// Mitsubishi GX Works2 project: LINEB-070924   PLC: Q26UDV

// task Task_01 (event TRUE, interval 0, priority 31): POU_01
// task temp_system (event TRUE, interval 0, priority 31): temp_system
// task comparater (event TRUE, interval 0, priority 31): comparater
// task Display (event TRUE, interval 0, priority 31): Display
// task cover_system (event TRUE, interval 0, priority 31): cover_system
// task input (event TRUE, interval 0, priority 31): input
// task output (event TRUE, interval 0, priority 31): output
// task payanak (event TRUE, interval 0, priority 31): 
// task pump_by_p_tongg (event TRUE, interval 0, priority 31): pump_by_p_tongg
// task rotation (event TRUE, interval 0, priority 31): rotation
// task lift (event TRUE, interval 0, priority 31): lift
// task blower (event TRUE, interval 0, priority 31): blower
// task carrier_move (event TRUE, interval 0, priority 31): carrier_move
// task door (event TRUE, interval 0, priority 31): door
// task lift_door_step (event TRUE, interval 0, priority 31): lift_door_step
// task Bit_Moniter_B (event TRUE, interval 0, priority 31): Bit_Moniter_B
// task input_conveyer (event TRUE, interval 0, priority 31): conveyer_input
// task coveyor_system (event TRUE, interval 0, priority 31): coveyor_system
// task convetor_output (event TRUE, interval 0, priority 31): conveyor_output
// task Scrubber (event TRUE, interval 0, priority 31): Scrubber
// task busket (event TRUE, interval 0, priority 31): busket
// task enter_line (event TRUE, interval 0, priority 31): enter_line
// task oven (event TRUE, interval 0, priority 31): oven
// task request_data (event TRUE, interval 0, priority 31): request_data
// task shower (event TRUE, interval 0, priority 31): shower
// task data_exchage (event TRUE, interval 0, priority 31): data_exchage
// task Alarm (event TRUE, interval 0, priority 31): Alarm
// task tower_lamp (event TRUE, interval 0, priority 31): tower_lamp
// task busker_step (event TRUE, interval 0, priority 31): busker_step
// task bit_monitor (event TRUE, interval 0, priority 31): bit_monitor
// task unload (event TRUE, interval 0, priority 31): unload
// task water_supply (event TRUE, interval 0, priority 31): water_supply
// task carrier_reset (event TRUE, interval 0, priority 31): carrier_reset
// task safty (event TRUE, interval 0, priority 31): safty
// task send_to_c (event TRUE, interval 0, priority 31): send_to_c
// task next_cap_step (event TRUE, interval 0, priority 31): next_cap_step
// task sent_to_c_key (event TRUE, interval 0, priority 31): sent_to_c_key
// task tank_time_B (event TRUE, interval 0, priority 31): tank_time_B
// task receive_c (event TRUE, interval 0, priority 31): receive_c
// task carrier_01 (event TRUE, interval 0, priority 31): carrier_01
// task carrier_02 (event TRUE, interval 0, priority 31): carrier_02
// task carrier_03 (event TRUE, interval 0, priority 31): carrier_03

PROGRAM Alarm
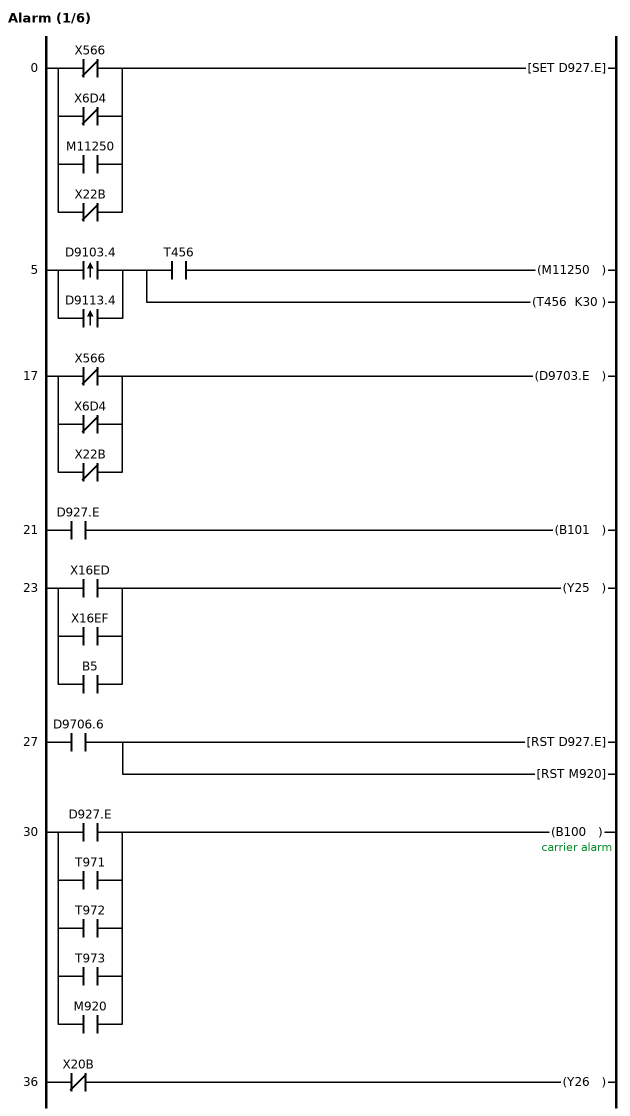
0     LDI     X566
      ORI     X6D4
      OR      M11250
      ORI     X22B
      SET     D927.E
5     LDP     D9103.4
      ORP     D9113.4
      MPS
      AND     T456
      OUT     M11250
      MPP
      OUT     T456 K30
17    LDI     X566
      ORI     X6D4
      ORI     X22B
      OUT     D9703.E
21    LD      D927.E
      OUT     B101
23    LD      X16ED
      OR      X16EF
      OR      B5
      OUT     Y25
27    LD      D9706.6
      RST     D927.E
      RST     M920
30    LD      D927.E
      OR      T971
      OR      T972
      OR      T973
      OR      M920
      OUT     B100  ; carrier alarm
36    LDI     X20B
      OUT     Y26
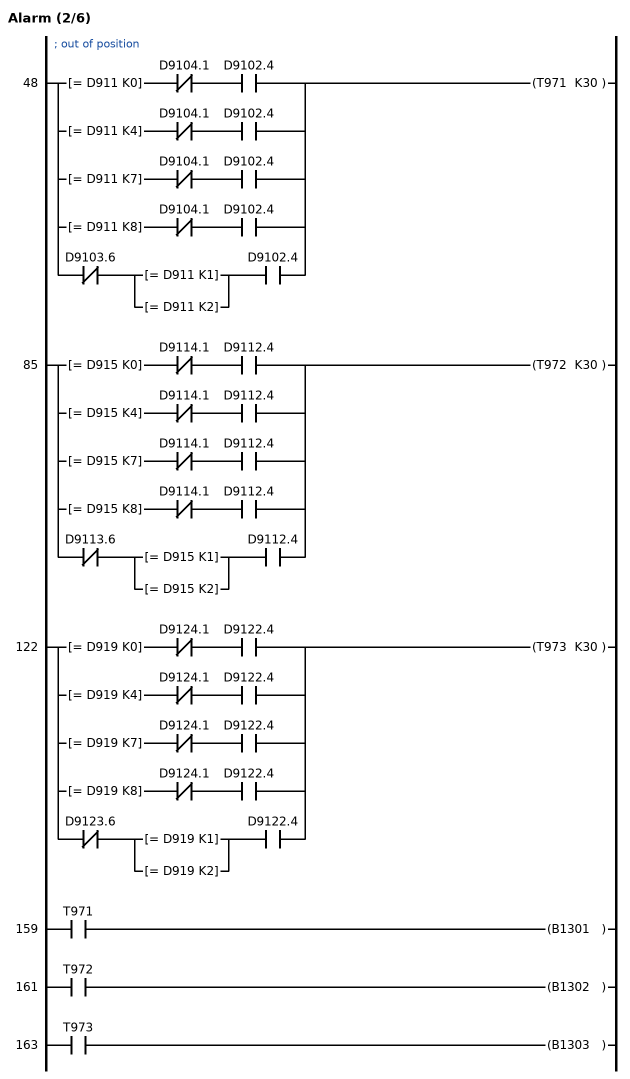
; out of position
48    LD=     D911 K0
      ANI     D9104.1
      AND     D9102.4
      LD=     D911 K4
      ANI     D9104.1
      AND     D9102.4
      ORB
      LD=     D911 K7
      ANI     D9104.1
      AND     D9102.4
      ORB
      LD=     D911 K8
      ANI     D9104.1
      AND     D9102.4
      ORB
      LDI     D9103.6
      LD=     D911 K1
      OR=     D911 K2
      ANB
      AND     D9102.4
      ORB
      OUT     T971 K30
85    LD=     D915 K0
      ANI     D9114.1
      AND     D9112.4
      LD=     D915 K4
      ANI     D9114.1
      AND     D9112.4
      ORB
      LD=     D915 K7
      ANI     D9114.1
      AND     D9112.4
      ORB
      LD=     D915 K8
      ANI     D9114.1
      AND     D9112.4
      ORB
      LDI     D9113.6
      LD=     D915 K1
      OR=     D915 K2
      ANB
      AND     D9112.4
      ORB
      OUT     T972 K30
122   LD=     D919 K0
      ANI     D9124.1
      AND     D9122.4
      LD=     D919 K4
      ANI     D9124.1
      AND     D9122.4
      ORB
      LD=     D919 K7
      ANI     D9124.1
      AND     D9122.4
      ORB
      LD=     D919 K8
      ANI     D9124.1
      AND     D9122.4
      ORB
      LDI     D9123.6
      LD=     D919 K1
      OR=     D919 K2
      ANB
      AND     D9122.4
      ORB
      OUT     T973 K30
159   LD      T971
      OUT     B1301
161   LD      T972
      OUT     B1302
163   LD      T973
      OUT     B1303
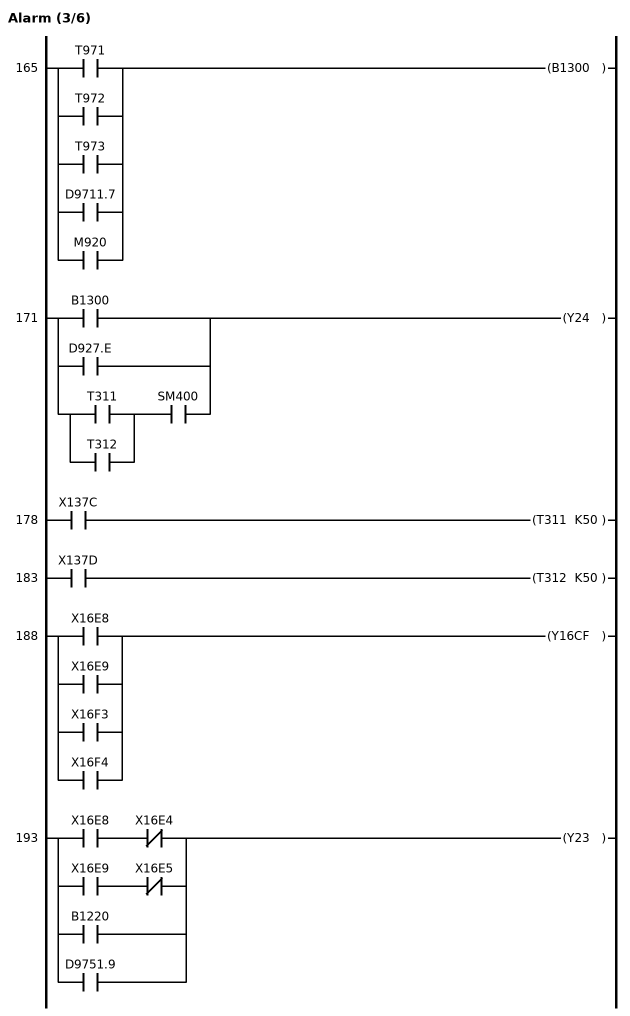
165   LD      T971
      OR      T972
      OR      T973
      OR      D9711.7
      OR      M920
      OUT     B1300
171   LD      B1300
      OR      D927.E
      LD      T311
      OR      T312
      AND     SM400
      ORB
      OUT     Y24
178   LD      X137C
      OUT     T311 K50
183   LD      X137D
      OUT     T312 K50
188   LD      X16E8
      OR      X16E9
      OR      X16F3
      OR      X16F4
      OUT     Y16CF
193   LD      X16E8
      ANI     X16E4
      LD      X16E9
      ANI     X16E5
      ORB
      OR      B1220
      OR      D9751.9
      OUT     Y23
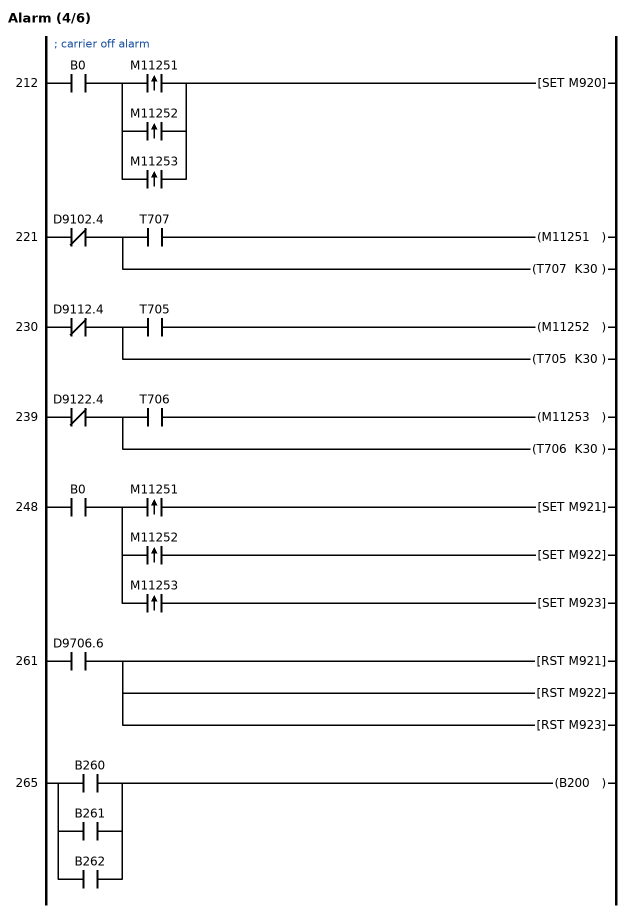
; carrier off alarm
212   LD      B0
      LDP     M11251
      ORP     M11252
      ORP     M11253
      ANB
      SET     M920
221   LDI     D9102.4
      MPS
      AND     T707
      OUT     M11251
      MPP
      OUT     T707 K30
230   LDI     D9112.4
      MPS
      AND     T705
      OUT     M11252
      MPP
      OUT     T705 K30
239   LDI     D9122.4
      MPS
      AND     T706
      OUT     M11253
      MPP
      OUT     T706 K30
248   LD      B0
      MPS
      ANDP    M11251
      SET     M921
      MRD
      ANDP    M11252
      SET     M922
      MPP
      ANDP    M11253
      SET     M923
261   LD      D9706.6
      RST     M921
      RST     M922
      RST     M923
265   LD      B260
      OR      B261
      OR      B262
      OUT     B200
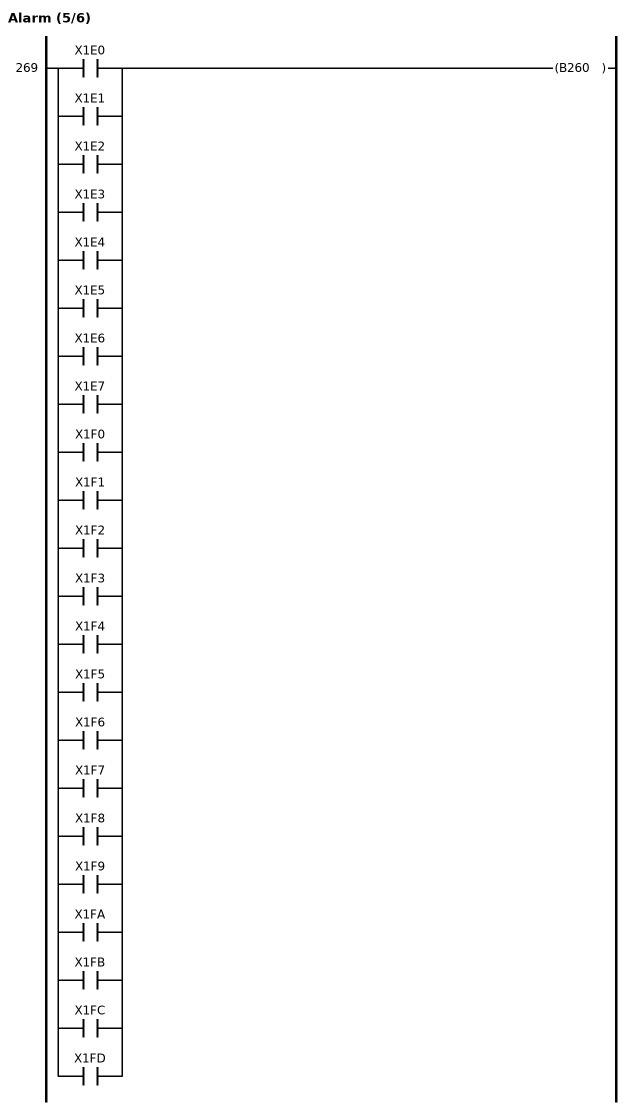
269   LD      X1E0
      OR      X1E1
      OR      X1E2
      OR      X1E3
      OR      X1E4
      OR      X1E5
      OR      X1E6
      OR      X1E7
      OR      X1F0
      OR      X1F1
      OR      X1F2
      OR      X1F3
      OR      X1F4
      OR      X1F5
      OR      X1F6
      OR      X1F7
      OR      X1F8
      OR      X1F9
      OR      X1FA
      OR      X1FB
      OR      X1FC
      OR      X1FD
      OUT     B260
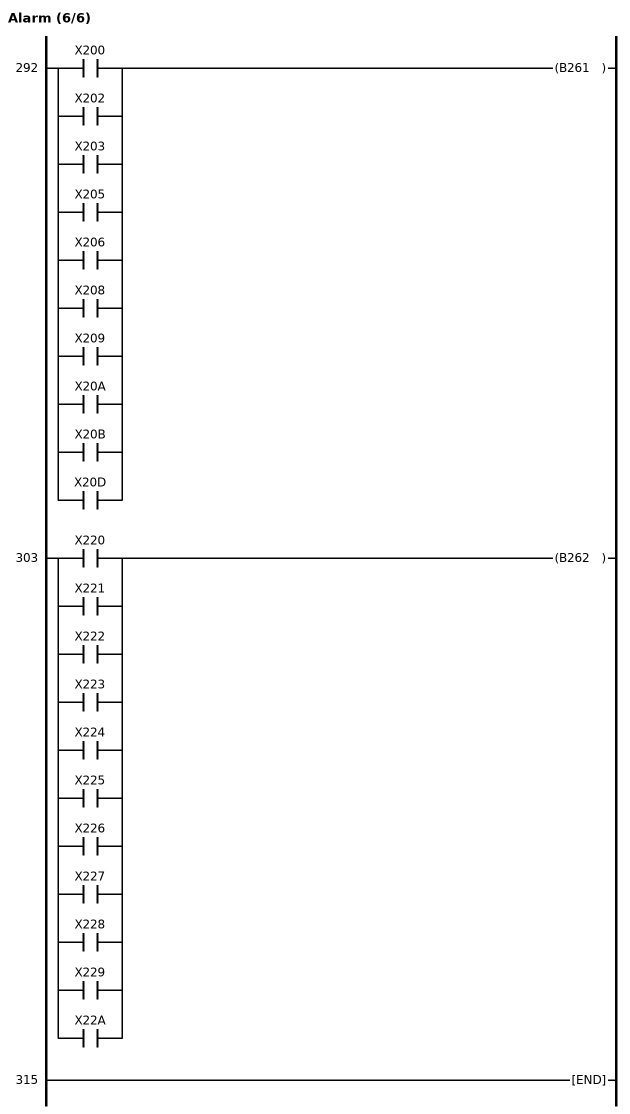
292   LD      X200
      OR      X202
      OR      X203
      OR      X205
      OR      X206
      OR      X208
      OR      X209
      OR      X20A
      OR      X20B
      OR      X20D
      OUT     B261
303   LD      X220
      OR      X221
      OR      X222
      OR      X223
      OR      X224
      OR      X225
      OR      X226
      OR      X227
      OR      X228
      OR      X229
      OR      X22A
      OUT     B262
315   END
END_PROGRAM

PROGRAM Bit_Moniter_B
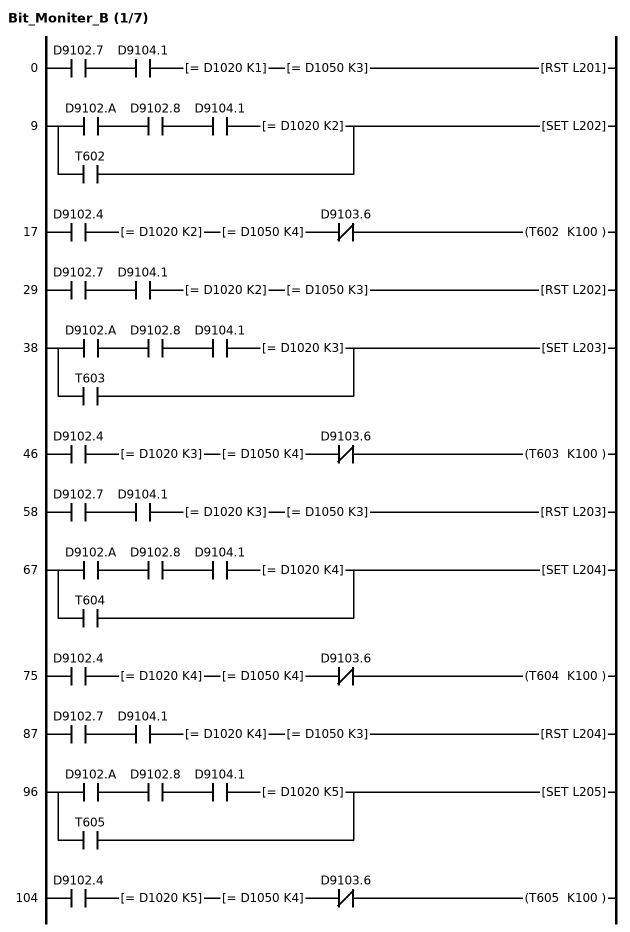
0     LD      D9102.7
      AND     D9104.1
      AND=    D1020 K1
      AND=    D1050 K3
      RST     L201
9     LD      D9102.A
      AND     D9102.8
      AND     D9104.1
      AND=    D1020 K2
      OR      T602
      SET     L202
17    LD      D9102.4
      AND=    D1020 K2
      AND=    D1050 K4
      ANI     D9103.6
      OUT     T602 K100
29    LD      D9102.7
      AND     D9104.1
      AND=    D1020 K2
      AND=    D1050 K3
      RST     L202
38    LD      D9102.A
      AND     D9102.8
      AND     D9104.1
      AND=    D1020 K3
      OR      T603
      SET     L203
46    LD      D9102.4
      AND=    D1020 K3
      AND=    D1050 K4
      ANI     D9103.6
      OUT     T603 K100
58    LD      D9102.7
      AND     D9104.1
      AND=    D1020 K3
      AND=    D1050 K3
      RST     L203
67    LD      D9102.A
      AND     D9102.8
      AND     D9104.1
      AND=    D1020 K4
      OR      T604
      SET     L204
75    LD      D9102.4
      AND=    D1020 K4
      AND=    D1050 K4
      ANI     D9103.6
      OUT     T604 K100
87    LD      D9102.7
      AND     D9104.1
      AND=    D1020 K4
      AND=    D1050 K3
      RST     L204
96    LD      D9102.A
      AND     D9102.8
      AND     D9104.1
      AND=    D1020 K5
      OR      T605
      SET     L205
104   LD      D9102.4
      AND=    D1020 K5
      AND=    D1050 K4
      ANI     D9103.6
      OUT     T605 K100
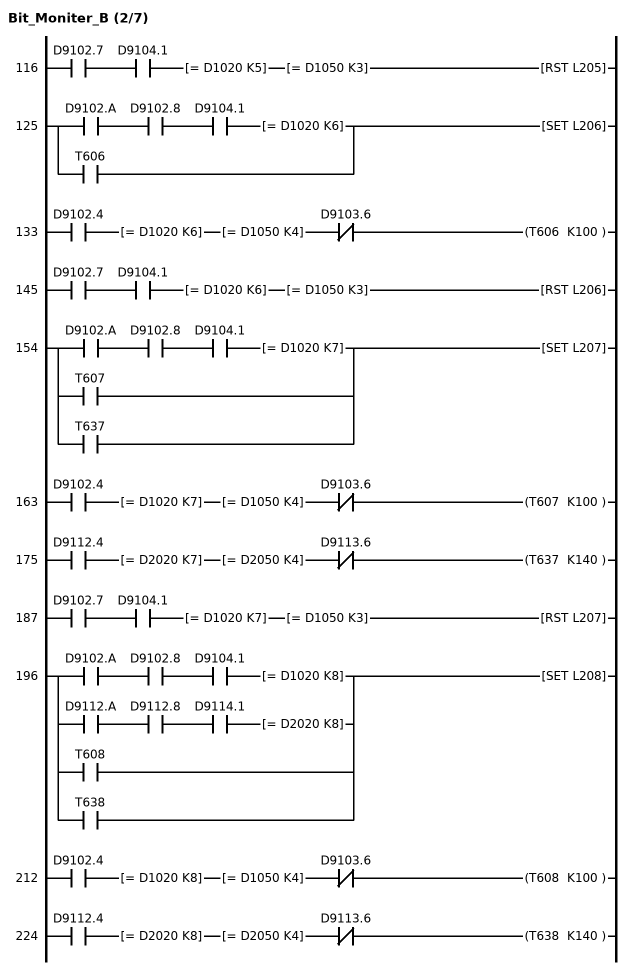
116   LD      D9102.7
      AND     D9104.1
      AND=    D1020 K5
      AND=    D1050 K3
      RST     L205
125   LD      D9102.A
      AND     D9102.8
      AND     D9104.1
      AND=    D1020 K6
      OR      T606
      SET     L206
133   LD      D9102.4
      AND=    D1020 K6
      AND=    D1050 K4
      ANI     D9103.6
      OUT     T606 K100
145   LD      D9102.7
      AND     D9104.1
      AND=    D1020 K6
      AND=    D1050 K3
      RST     L206
154   LD      D9102.A
      AND     D9102.8
      AND     D9104.1
      AND=    D1020 K7
      OR      T607
      OR      T637
      SET     L207
163   LD      D9102.4
      AND=    D1020 K7
      AND=    D1050 K4
      ANI     D9103.6
      OUT     T607 K100
175   LD      D9112.4
      AND=    D2020 K7
      AND=    D2050 K4
      ANI     D9113.6
      OUT     T637 K140
187   LD      D9102.7
      AND     D9104.1
      AND=    D1020 K7
      AND=    D1050 K3
      RST     L207
196   LD      D9102.A
      AND     D9102.8
      AND     D9104.1
      AND=    D1020 K8
      LD      D9112.A
      AND     D9112.8
      AND     D9114.1
      AND=    D2020 K8
      ORB
      OR      T608
      OR      T638
      SET     L208
212   LD      D9102.4
      AND=    D1020 K8
      AND=    D1050 K4
      ANI     D9103.6
      OUT     T608 K100
224   LD      D9112.4
      AND=    D2020 K8
      AND=    D2050 K4
      ANI     D9113.6
      OUT     T638 K140
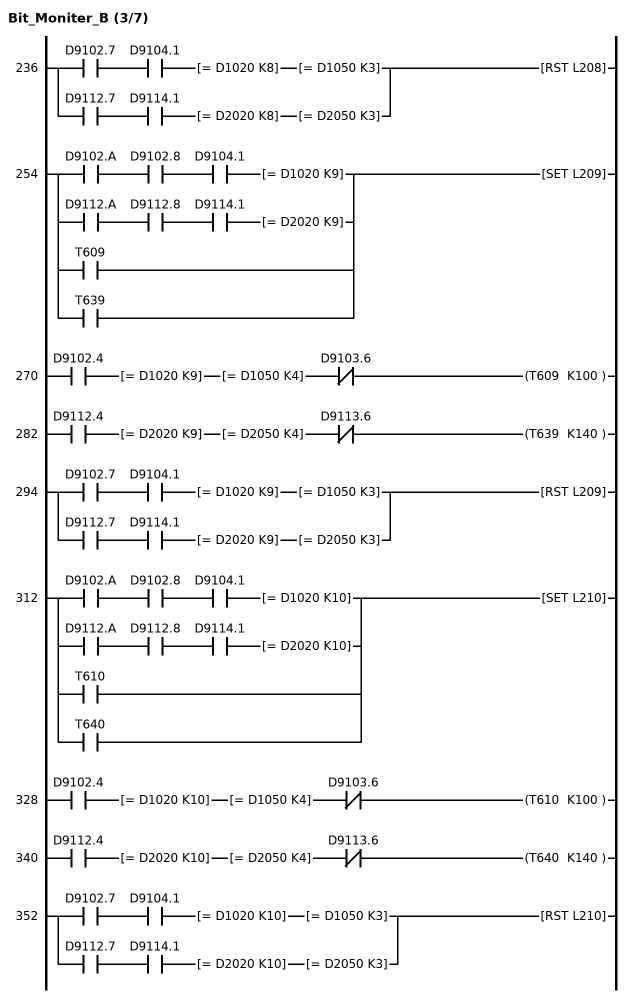
236   LD      D9102.7
      AND     D9104.1
      AND=    D1020 K8
      AND=    D1050 K3
      LD      D9112.7
      AND     D9114.1
      AND=    D2020 K8
      AND=    D2050 K3
      ORB
      RST     L208
254   LD      D9102.A
      AND     D9102.8
      AND     D9104.1
      AND=    D1020 K9
      LD      D9112.A
      AND     D9112.8
      AND     D9114.1
      AND=    D2020 K9
      ORB
      OR      T609
      OR      T639
      SET     L209
270   LD      D9102.4
      AND=    D1020 K9
      AND=    D1050 K4
      ANI     D9103.6
      OUT     T609 K100
282   LD      D9112.4
      AND=    D2020 K9
      AND=    D2050 K4
      ANI     D9113.6
      OUT     T639 K140
294   LD      D9102.7
      AND     D9104.1
      AND=    D1020 K9
      AND=    D1050 K3
      LD      D9112.7
      AND     D9114.1
      AND=    D2020 K9
      AND=    D2050 K3
      ORB
      RST     L209
312   LD      D9102.A
      AND     D9102.8
      AND     D9104.1
      AND=    D1020 K10
      LD      D9112.A
      AND     D9112.8
      AND     D9114.1
      AND=    D2020 K10
      ORB
      OR      T610
      OR      T640
      SET     L210
328   LD      D9102.4
      AND=    D1020 K10
      AND=    D1050 K4
      ANI     D9103.6
      OUT     T610 K100
340   LD      D9112.4
      AND=    D2020 K10
      AND=    D2050 K4
      ANI     D9113.6
      OUT     T640 K140
352   LD      D9102.7
      AND     D9104.1
      AND=    D1020 K10
      AND=    D1050 K3
      LD      D9112.7
      AND     D9114.1
      AND=    D2020 K10
      AND=    D2050 K3
      ORB
      RST     L210
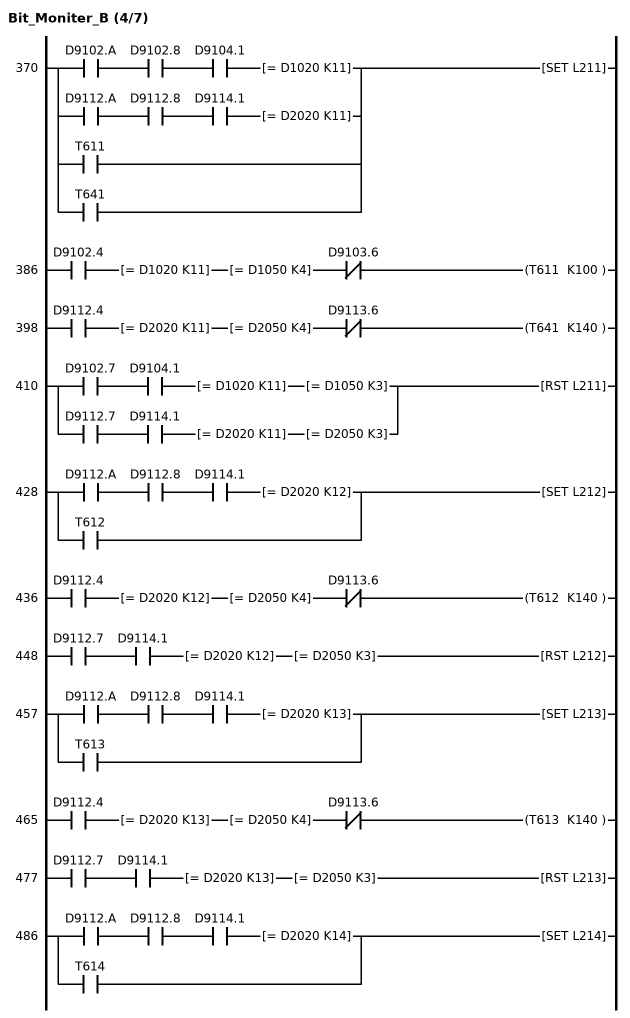
370   LD      D9102.A
      AND     D9102.8
      AND     D9104.1
      AND=    D1020 K11
      LD      D9112.A
      AND     D9112.8
      AND     D9114.1
      AND=    D2020 K11
      ORB
      OR      T611
      OR      T641
      SET     L211
386   LD      D9102.4
      AND=    D1020 K11
      AND=    D1050 K4
      ANI     D9103.6
      OUT     T611 K100
398   LD      D9112.4
      AND=    D2020 K11
      AND=    D2050 K4
      ANI     D9113.6
      OUT     T641 K140
410   LD      D9102.7
      AND     D9104.1
      AND=    D1020 K11
      AND=    D1050 K3
      LD      D9112.7
      AND     D9114.1
      AND=    D2020 K11
      AND=    D2050 K3
      ORB
      RST     L211
428   LD      D9112.A
      AND     D9112.8
      AND     D9114.1
      AND=    D2020 K12
      OR      T612
      SET     L212
436   LD      D9112.4
      AND=    D2020 K12
      AND=    D2050 K4
      ANI     D9113.6
      OUT     T612 K140
448   LD      D9112.7
      AND     D9114.1
      AND=    D2020 K12
      AND=    D2050 K3
      RST     L212
457   LD      D9112.A
      AND     D9112.8
      AND     D9114.1
      AND=    D2020 K13
      OR      T613
      SET     L213
465   LD      D9112.4
      AND=    D2020 K13
      AND=    D2050 K4
      ANI     D9113.6
      OUT     T613 K140
477   LD      D9112.7
      AND     D9114.1
      AND=    D2020 K13
      AND=    D2050 K3
      RST     L213
486   LD      D9112.A
      AND     D9112.8
      AND     D9114.1
      AND=    D2020 K14
      OR      T614
      SET     L214
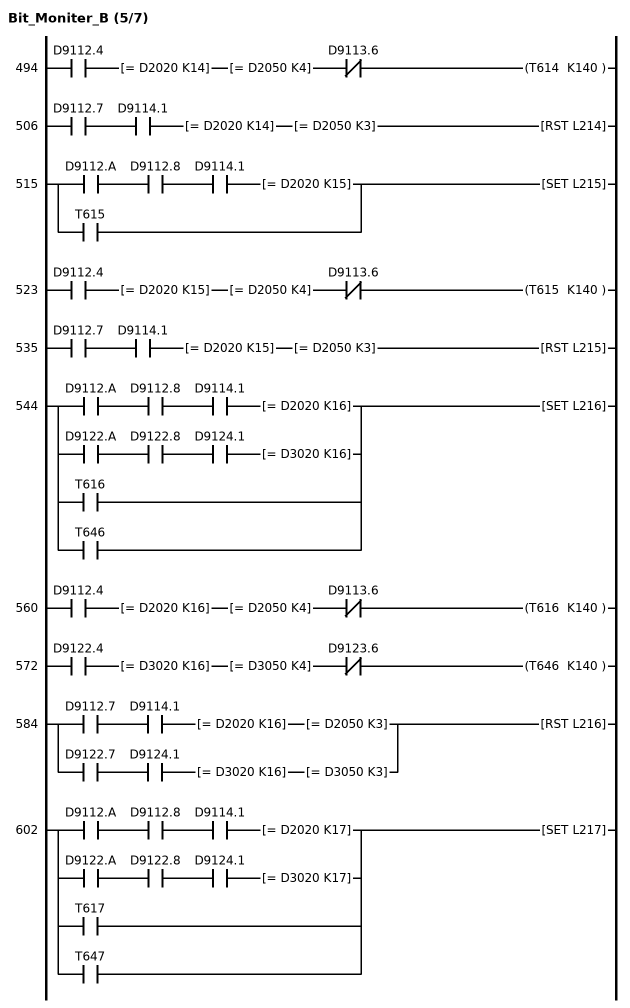
494   LD      D9112.4
      AND=    D2020 K14
      AND=    D2050 K4
      ANI     D9113.6
      OUT     T614 K140
506   LD      D9112.7
      AND     D9114.1
      AND=    D2020 K14
      AND=    D2050 K3
      RST     L214
515   LD      D9112.A
      AND     D9112.8
      AND     D9114.1
      AND=    D2020 K15
      OR      T615
      SET     L215
523   LD      D9112.4
      AND=    D2020 K15
      AND=    D2050 K4
      ANI     D9113.6
      OUT     T615 K140
535   LD      D9112.7
      AND     D9114.1
      AND=    D2020 K15
      AND=    D2050 K3
      RST     L215
544   LD      D9112.A
      AND     D9112.8
      AND     D9114.1
      AND=    D2020 K16
      LD      D9122.A
      AND     D9122.8
      AND     D9124.1
      AND=    D3020 K16
      ORB
      OR      T616
      OR      T646
      SET     L216
560   LD      D9112.4
      AND=    D2020 K16
      AND=    D2050 K4
      ANI     D9113.6
      OUT     T616 K140
572   LD      D9122.4
      AND=    D3020 K16
      AND=    D3050 K4
      ANI     D9123.6
      OUT     T646 K140
584   LD      D9112.7
      AND     D9114.1
      AND=    D2020 K16
      AND=    D2050 K3
      LD      D9122.7
      AND     D9124.1
      AND=    D3020 K16
      AND=    D3050 K3
      ORB
      RST     L216
602   LD      D9112.A
      AND     D9112.8
      AND     D9114.1
      AND=    D2020 K17
      LD      D9122.A
      AND     D9122.8
      AND     D9124.1
      AND=    D3020 K17
      ORB
      OR      T617
      OR      T647
      SET     L217
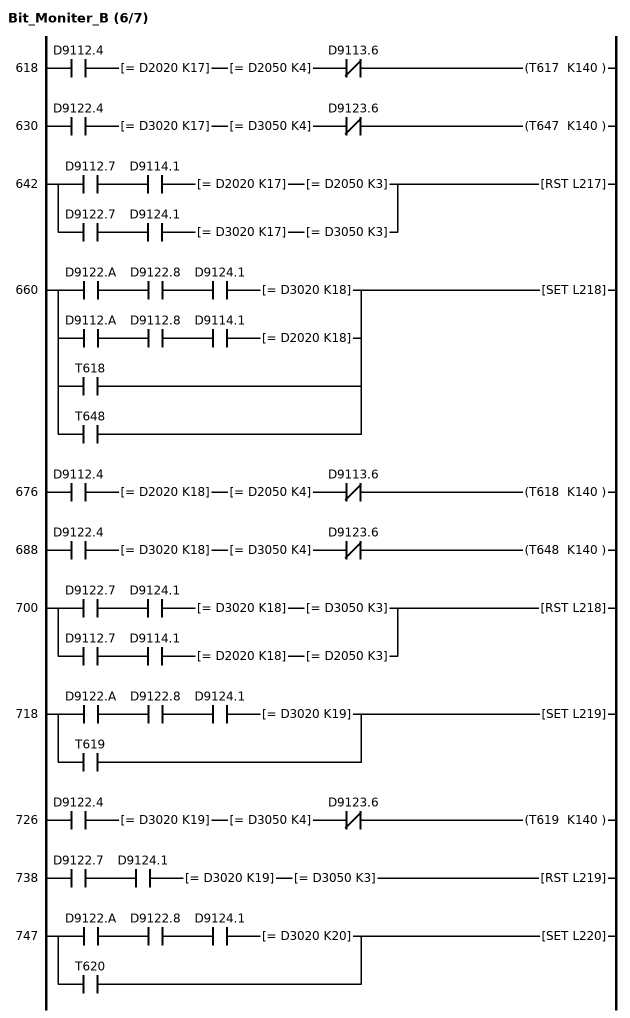
618   LD      D9112.4
      AND=    D2020 K17
      AND=    D2050 K4
      ANI     D9113.6
      OUT     T617 K140
630   LD      D9122.4
      AND=    D3020 K17
      AND=    D3050 K4
      ANI     D9123.6
      OUT     T647 K140
642   LD      D9112.7
      AND     D9114.1
      AND=    D2020 K17
      AND=    D2050 K3
      LD      D9122.7
      AND     D9124.1
      AND=    D3020 K17
      AND=    D3050 K3
      ORB
      RST     L217
660   LD      D9122.A
      AND     D9122.8
      AND     D9124.1
      AND=    D3020 K18
      LD      D9112.A
      AND     D9112.8
      AND     D9114.1
      AND=    D2020 K18
      ORB
      OR      T618
      OR      T648
      SET     L218
676   LD      D9112.4
      AND=    D2020 K18
      AND=    D2050 K4
      ANI     D9113.6
      OUT     T618 K140
688   LD      D9122.4
      AND=    D3020 K18
      AND=    D3050 K4
      ANI     D9123.6
      OUT     T648 K140
700   LD      D9122.7
      AND     D9124.1
      AND=    D3020 K18
      AND=    D3050 K3
      LD      D9112.7
      AND     D9114.1
      AND=    D2020 K18
      AND=    D2050 K3
      ORB
      RST     L218
718   LD      D9122.A
      AND     D9122.8
      AND     D9124.1
      AND=    D3020 K19
      OR      T619
      SET     L219
726   LD      D9122.4
      AND=    D3020 K19
      AND=    D3050 K4
      ANI     D9123.6
      OUT     T619 K140
738   LD      D9122.7
      AND     D9124.1
      AND=    D3020 K19
      AND=    D3050 K3
      RST     L219
747   LD      D9122.A
      AND     D9122.8
      AND     D9124.1
      AND=    D3020 K20
      OR      T620
      SET     L220
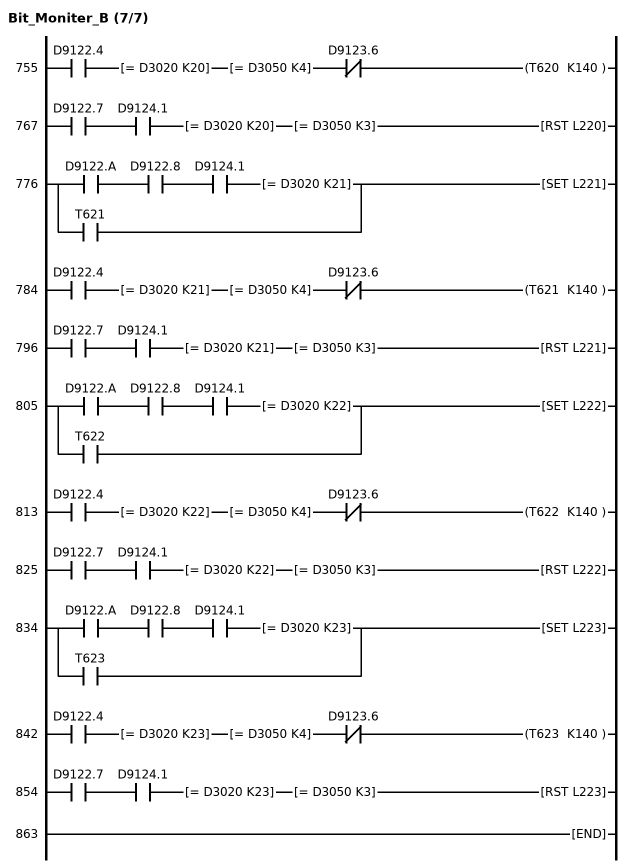
755   LD      D9122.4
      AND=    D3020 K20
      AND=    D3050 K4
      ANI     D9123.6
      OUT     T620 K140
767   LD      D9122.7
      AND     D9124.1
      AND=    D3020 K20
      AND=    D3050 K3
      RST     L220
776   LD      D9122.A
      AND     D9122.8
      AND     D9124.1
      AND=    D3020 K21
      OR      T621
      SET     L221
784   LD      D9122.4
      AND=    D3020 K21
      AND=    D3050 K4
      ANI     D9123.6
      OUT     T621 K140
796   LD      D9122.7
      AND     D9124.1
      AND=    D3020 K21
      AND=    D3050 K3
      RST     L221
805   LD      D9122.A
      AND     D9122.8
      AND     D9124.1
      AND=    D3020 K22
      OR      T622
      SET     L222
813   LD      D9122.4
      AND=    D3020 K22
      AND=    D3050 K4
      ANI     D9123.6
      OUT     T622 K140
825   LD      D9122.7
      AND     D9124.1
      AND=    D3020 K22
      AND=    D3050 K3
      RST     L222
834   LD      D9122.A
      AND     D9122.8
      AND     D9124.1
      AND=    D3020 K23
      OR      T623
      SET     L223
842   LD      D9122.4
      AND=    D3020 K23
      AND=    D3050 K4
      ANI     D9123.6
      OUT     T623 K140
854   LD      D9122.7
      AND     D9124.1
      AND=    D3020 K23
      AND=    D3050 K3
      RST     L223
863   END
END_PROGRAM

PROGRAM bit_monitor
0     END
END_PROGRAM

PROGRAM blower
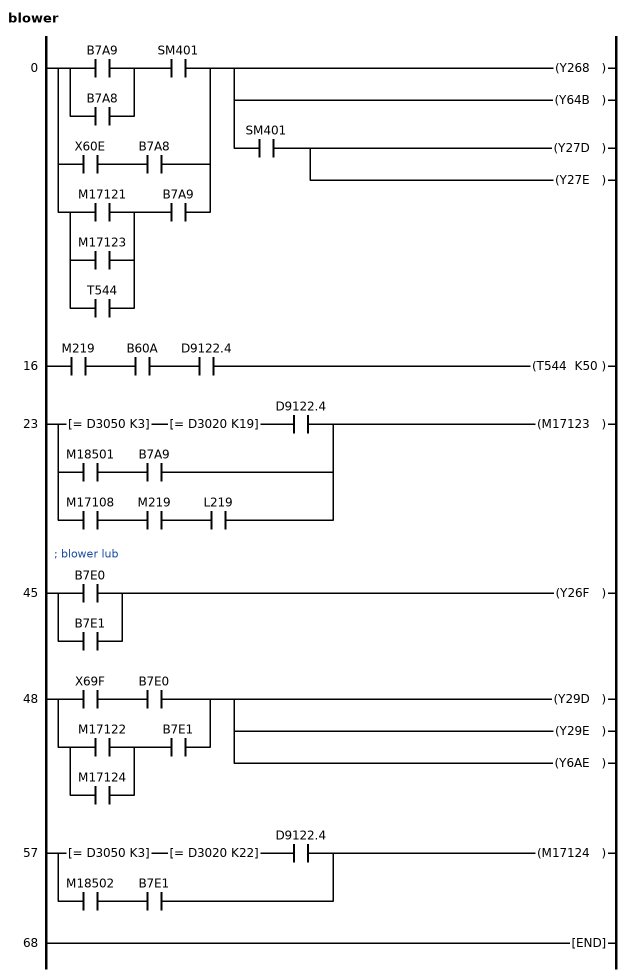
0     LD      B7A9
      OR      B7A8
      AND     SM401
      LD      X60E
      AND     B7A8
      ORB
      LD      M17121
      OR      M17123
      OR      T544
      AND     B7A9
      ORB
      OUT     Y268
      OUT     Y64B
      AND     SM401
      OUT     Y27D
      OUT     Y27E
16    LD      M219
      AND     B60A
      AND     D9122.4
      OUT     T544 K50
23    LD=     D3050 K3
      AND=    D3020 K19
      AND     D9122.4
      LD      M18501
      AND     B7A9
      ORB
      LD      M17108
      AND     M219
      AND     L219
      ORB
      OUT     M17123
; blower lub
45    LD      B7E0
      OR      B7E1
      OUT     Y26F
48    LD      X69F
      AND     B7E0
      LD      M17122
      OR      M17124
      AND     B7E1
      ORB
      OUT     Y29D
      OUT     Y29E
      OUT     Y6AE
57    LD=     D3050 K3
      AND=    D3020 K22
      AND     D9122.4
      LD      M18502
      AND     B7E1
      ORB
      OUT     M17124
68    END
END_PROGRAM

PROGRAM busker_step
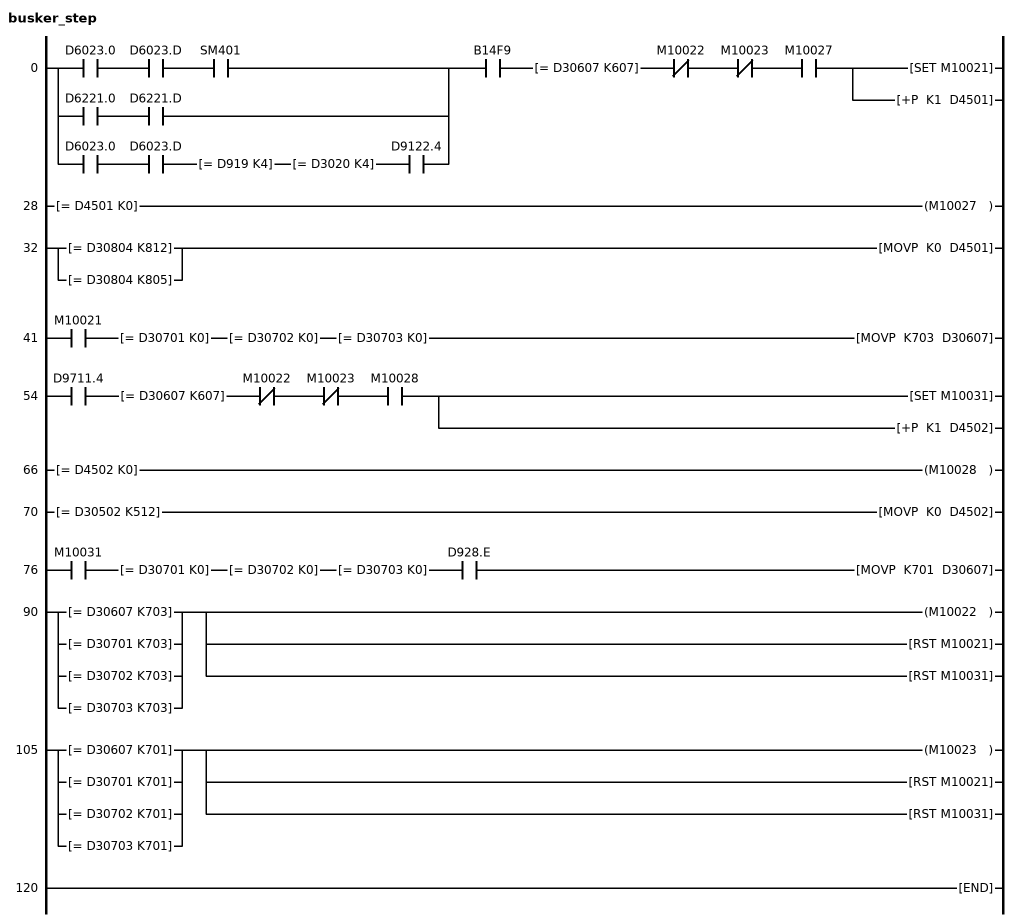
0     LD      D6023.0
      AND     D6023.D
      AND     SM401
      LD      D6221.0
      AND     D6221.D
      ORB
      LD      D6023.0
      AND     D6023.D
      AND=    D919 K4
      AND=    D3020 K4
      AND     D9122.4
      ORB
      AND     B14F9
      AND=    D30607 K607
      ANI     M10022
      ANI     M10023
      AND     M10027
      SET     M10021
      +P      K1 D4501
28    LD=     D4501 K0
      OUT     M10027
32    LD=     D30804 K812
      OR=     D30804 K805
      MOVP    K0 D4501
41    LD      M10021
      AND=    D30701 K0
      AND=    D30702 K0
      AND=    D30703 K0
      MOVP    K703 D30607
54    LD      D9711.4
      AND=    D30607 K607
      ANI     M10022
      ANI     M10023
      AND     M10028
      SET     M10031
      +P      K1 D4502
66    LD=     D4502 K0
      OUT     M10028
70    LD=     D30502 K512
      MOVP    K0 D4502
76    LD      M10031
      AND=    D30701 K0
      AND=    D30702 K0
      AND=    D30703 K0
      AND     D928.E
      MOVP    K701 D30607
90    LD=     D30607 K703
      OR=     D30701 K703
      OR=     D30702 K703
      OR=     D30703 K703
      OUT     M10022
      RST     M10021
      RST     M10031
105   LD=     D30607 K701
      OR=     D30701 K701
      OR=     D30702 K701
      OR=     D30703 K701
      OUT     M10023
      RST     M10021
      RST     M10031
120   END
END_PROGRAM

PROGRAM busket
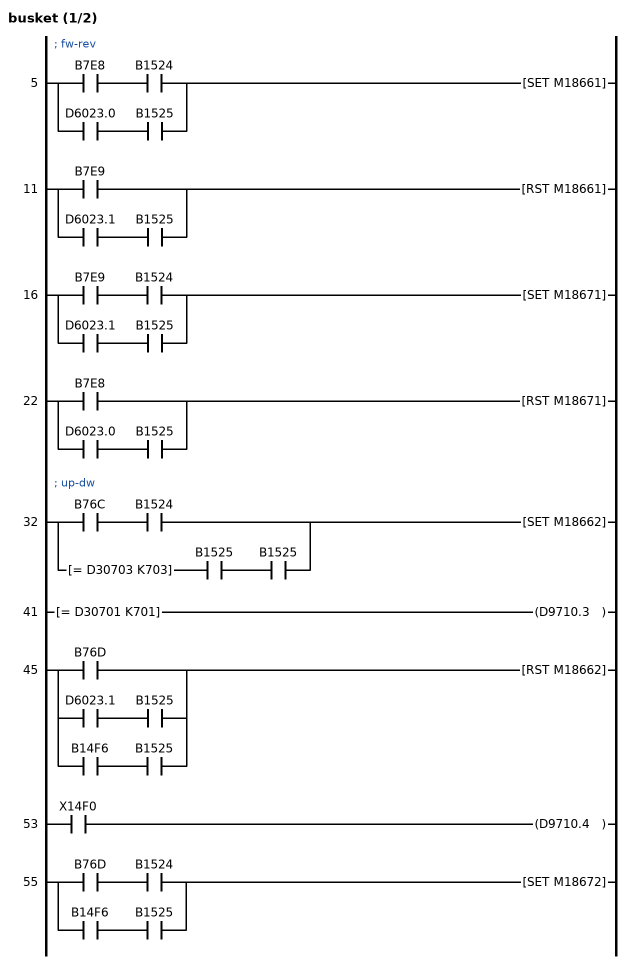
; fw-rev
5     LD      B7E8
      AND     B1524
      LD      D6023.0
      AND     B1525
      ORB
      SET     M18661
11    LD      B7E9
      LD      D6023.1
      AND     B1525
      ORB
      RST     M18661
16    LD      B7E9
      AND     B1524
      LD      D6023.1
      AND     B1525
      ORB
      SET     M18671
22    LD      B7E8
      LD      D6023.0
      AND     B1525
      ORB
      RST     M18671
; up-dw
32    LD      B76C
      AND     B1524
      LD=     D30703 K703
      AND     B1525
      AND     B1525
      ORB
      SET     M18662
41    LD=     D30701 K701
      OUT     D9710.3
45    LD      B76D
      LD      D6023.1
      AND     B1525
      ORB
      LD      B14F6
      AND     B1525
      ORB
      RST     M18662
53    LD      X14F0
      OUT     D9710.4
55    LD      B76D
      AND     B1524
      LD      B14F6
      AND     B1525
      ORB
      SET     M18672
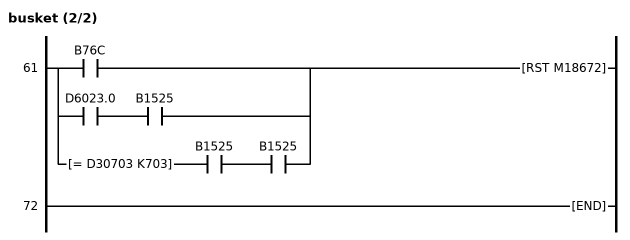
61    LD      B76C
      LD      D6023.0
      AND     B1525
      ORB
      LD=     D30703 K703
      AND     B1525
      AND     B1525
      ORB
      RST     M18672
72    END
END_PROGRAM

FUNCTION_BLOCK c_comm_1
VAR_INPUT
  P1_input : INT;
  P2_input : INT;
  P3_input : INT;
END_VAR
VAR_IN_OUT
  step_on : INT;
END_VAR
VAR_INPUT
  position : INT;
END_VAR
VAR
  p2_buff : INT;
END_VAR
VAR_OUTPUT
  P1_output : INT;
  P2_output : INT;
  P3_output : INT;
END_VAR
VAR_IN_OUT
  end_step_01 : INT;
END_VAR
VAR_OUTPUT
  end_signal : BOOL;
END_VAR
VAR
  mc_1234 : BOOL;
  line1_10_buff : INT;
  line2_10_buff : INT;
END_VAR
VAR_OUTPUT
  next_signal : BOOL;
END_VAR
VAR
  next_signal_01 : BOOL;
  next_signal_03 : BOOL;
  next_signal_04 : BOOL;
  next_signal_05 : BOOL;
  next_signal_06 : BOOL;
  next_signal_07 : BOOL;
  next_signal_08 : BOOL;
  punch1 : BOOL;
  punch3 : BOOL;
  punch4 : BOOL;
  punch5 : BOOL;
  punch6 : BOOL;
  punch7 : BOOL;
END_VAR
VAR_OUTPUT
  punch : BOOL;
END_VAR
VAR
  punch2 : BOOL;
  timee : TIMER;
  timee2 : TIMER;
  timee3 : TIMER;
END_VAR
VAR_INPUT
  d40wait : INT;
END_VAR
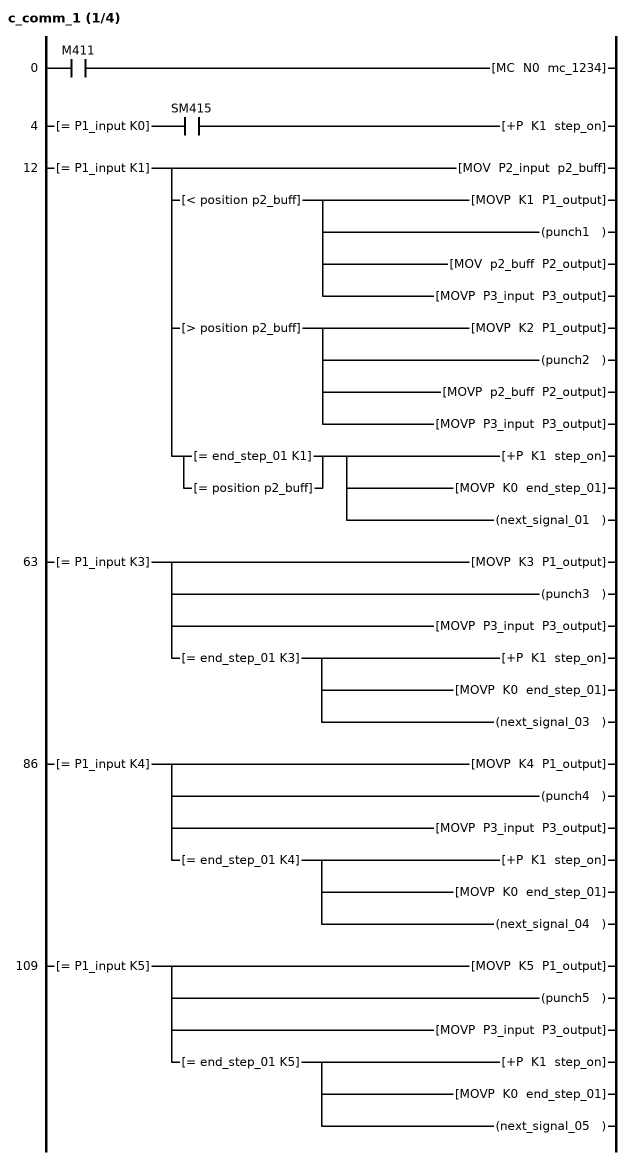
0     LD      M411
      MC      N0 mc_1234
4     LD=     P1_input K0
      AND     SM415
      +P      K1 step_on
12    LD=     P1_input K1
      MOV     P2_input p2_buff
      MPS
      AND<    position p2_buff
      MOVP    K1 P1_output
      OUT     punch1
      MOV     p2_buff P2_output
      MOVP    P3_input P3_output
      MRD
      AND>    position p2_buff
      MOVP    K2 P1_output
      OUT     punch2
      MOVP    p2_buff P2_output
      MOVP    P3_input P3_output
      MPP
      LD=     end_step_01 K1
      OR=     position p2_buff
      ANB
      +P      K1 step_on
      MOVP    K0 end_step_01
      OUT     next_signal_01
63    LD=     P1_input K3
      MOVP    K3 P1_output
      OUT     punch3
      MOVP    P3_input P3_output
      AND=    end_step_01 K3
      +P      K1 step_on
      MOVP    K0 end_step_01
      OUT     next_signal_03
86    LD=     P1_input K4
      MOVP    K4 P1_output
      OUT     punch4
      MOVP    P3_input P3_output
      AND=    end_step_01 K4
      +P      K1 step_on
      MOVP    K0 end_step_01
      OUT     next_signal_04
109   LD=     P1_input K5
      MOVP    K5 P1_output
      OUT     punch5
      MOVP    P3_input P3_output
      AND=    end_step_01 K5
      +P      K1 step_on
      MOVP    K0 end_step_01
      OUT     next_signal_05
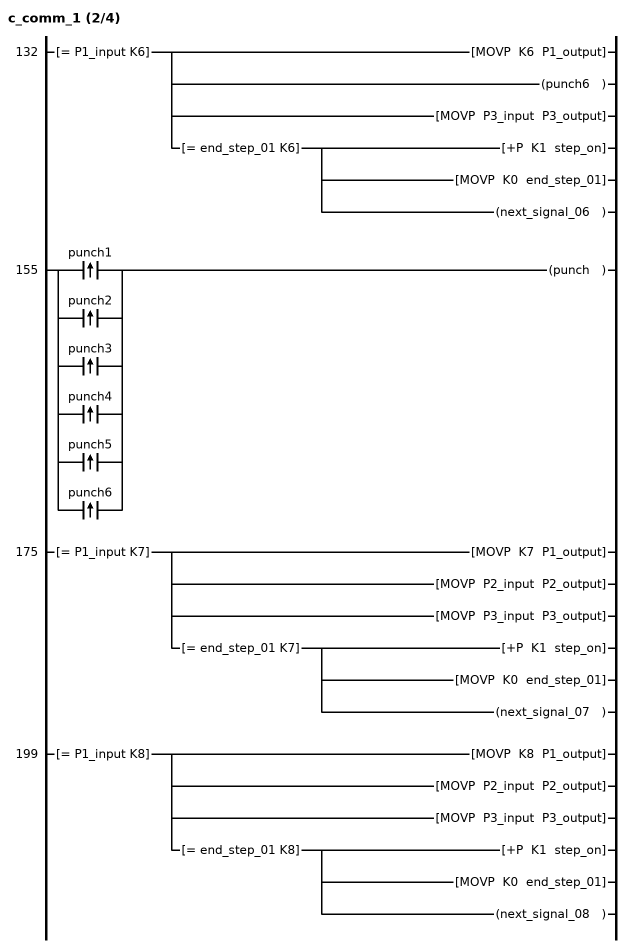
132   LD=     P1_input K6
      MOVP    K6 P1_output
      OUT     punch6
      MOVP    P3_input P3_output
      AND=    end_step_01 K6
      +P      K1 step_on
      MOVP    K0 end_step_01
      OUT     next_signal_06
155   LDP     punch1
      ORP     punch2
      ORP     punch3
      ORP     punch4
      ORP     punch5
      ORP     punch6
      OUT     punch
175   LD=     P1_input K7
      MOVP    K7 P1_output
      MOVP    P2_input P2_output
      MOVP    P3_input P3_output
      AND=    end_step_01 K7
      +P      K1 step_on
      MOVP    K0 end_step_01
      OUT     next_signal_07
199   LD=     P1_input K8
      MOVP    K8 P1_output
      MOVP    P2_input P2_output
      MOVP    P3_input P3_output
      AND=    end_step_01 K8
      +P      K1 step_on
      MOVP    K0 end_step_01
      OUT     next_signal_08
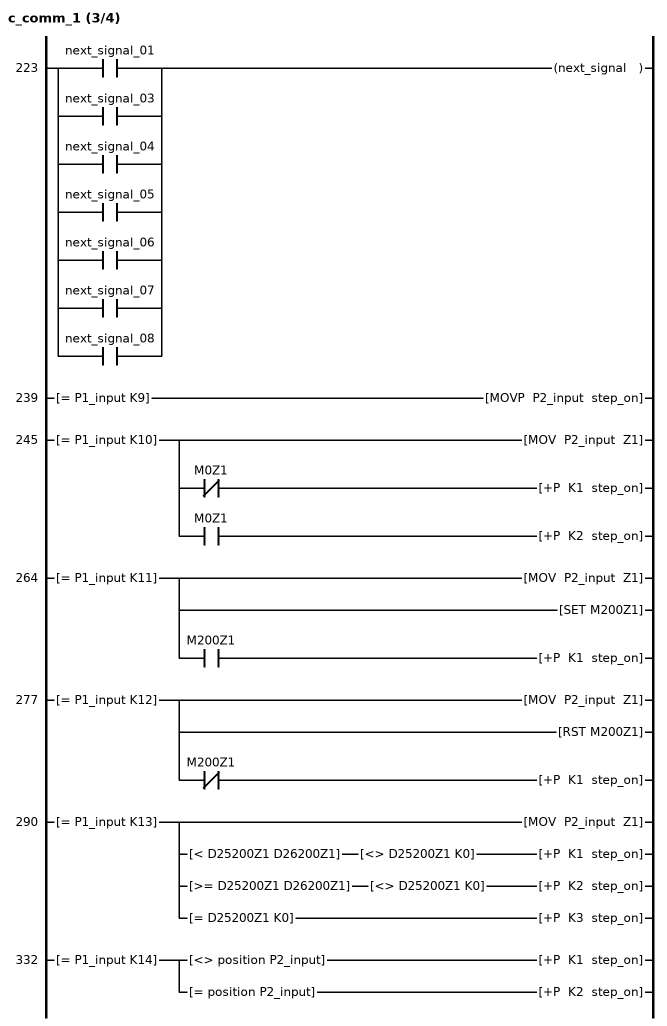
223   LD      next_signal_01
      OR      next_signal_03
      OR      next_signal_04
      OR      next_signal_05
      OR      next_signal_06
      OR      next_signal_07
      OR      next_signal_08
      OUT     next_signal
239   LD=     P1_input K9
      MOVP    P2_input step_on
245   LD=     P1_input K10
      MOV     P2_input Z1
      MPS
      ANI     M0Z1
      +P      K1 step_on
      MPP
      AND     M0Z1
      +P      K2 step_on
264   LD=     P1_input K11
      MOV     P2_input Z1
      SET     M200Z1
      AND     M200Z1
      +P      K1 step_on
277   LD=     P1_input K12
      MOV     P2_input Z1
      RST     M200Z1
      ANI     M200Z1
      +P      K1 step_on
290   LD=     P1_input K13
      MOV     P2_input Z1
      MPS
      AND<    D25200Z1 D26200Z1
      AND<>   D25200Z1 K0
      +P      K1 step_on
      MRD
      AND>=   D25200Z1 D26200Z1
      AND<>   D25200Z1 K0
      +P      K2 step_on
      MPP
      AND=    D25200Z1 K0
      +P      K3 step_on
332   LD=     P1_input K14
      MPS
      AND<>   position P2_input
      +P      K1 step_on
      MPP
      AND=    position P2_input
      +P      K2 step_on
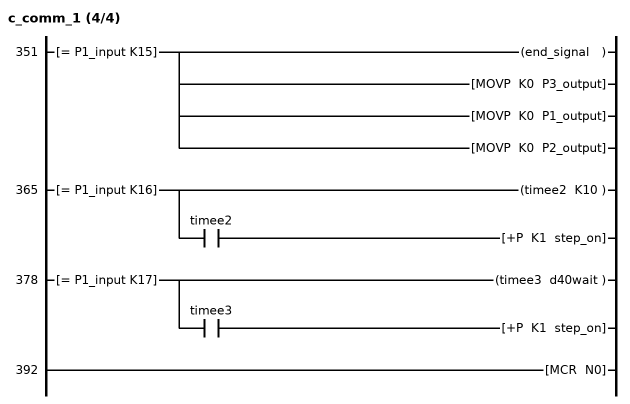
351   LD=     P1_input K15
      OUT     end_signal
      MOVP    K0 P3_output
      MOVP    K0 P1_output
      MOVP    K0 P2_output
365   LD=     P1_input K16
      OUT     timee2 K10
      AND     timee2
      +P      K1 step_on
378   LD=     P1_input K17
      OUT     timee3 d40wait
      AND     timee3
      +P      K1 step_on
392   MCR     N0
END_FUNCTION_BLOCK

FUNCTION_BLOCK c_comm_2
VAR_INPUT
  P1_input : INT;
  P2_input : INT;
  P3_input : INT;
END_VAR
VAR_IN_OUT
  step_on : INT;
END_VAR
VAR_INPUT
  position : INT;
END_VAR
VAR
  p2_buff : INT;
END_VAR
VAR_OUTPUT
  P1_output : INT;
  P2_output : INT;
  P3_output : INT;
END_VAR
VAR_IN_OUT
  end_step_01 : INT;
END_VAR
VAR_OUTPUT
  end_signal : BOOL;
END_VAR
VAR
  mc_1234 : BOOL;
  line1_10_buff : INT;
  line2_10_buff : INT;
END_VAR
VAR_OUTPUT
  next_signal : BOOL;
END_VAR
VAR
  next_signal_01 : BOOL;
  next_signal_03 : BOOL;
  next_signal_04 : BOOL;
  next_signal_05 : BOOL;
  next_signal_06 : BOOL;
  next_signal_07 : BOOL;
  next_signal_08 : BOOL;
  punch1 : BOOL;
  punch3 : BOOL;
  punch4 : BOOL;
  punch5 : BOOL;
  punch6 : BOOL;
  punch7 : BOOL;
END_VAR
VAR_OUTPUT
  punch : BOOL;
END_VAR
VAR
  punch2 : BOOL;
  timee : TIMER;
  timee2 : TIMER;
END_VAR
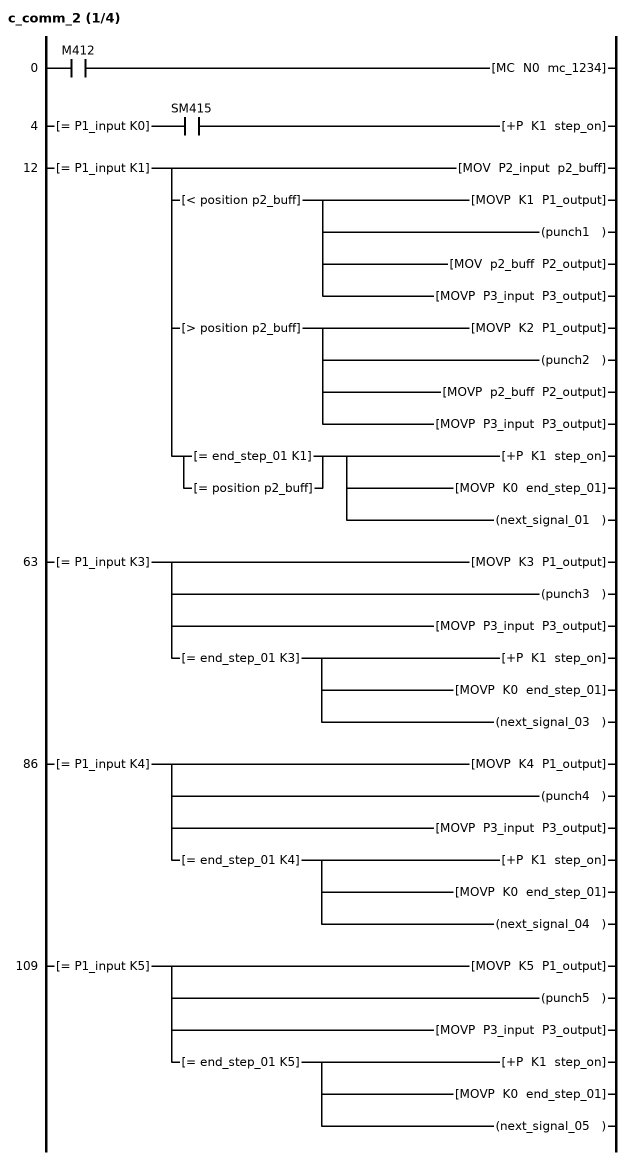
0     LD      M412
      MC      N0 mc_1234
4     LD=     P1_input K0
      AND     SM415
      +P      K1 step_on
12    LD=     P1_input K1
      MOV     P2_input p2_buff
      MPS
      AND<    position p2_buff
      MOVP    K1 P1_output
      OUT     punch1
      MOV     p2_buff P2_output
      MOVP    P3_input P3_output
      MRD
      AND>    position p2_buff
      MOVP    K2 P1_output
      OUT     punch2
      MOVP    p2_buff P2_output
      MOVP    P3_input P3_output
      MPP
      LD=     end_step_01 K1
      OR=     position p2_buff
      ANB
      +P      K1 step_on
      MOVP    K0 end_step_01
      OUT     next_signal_01
63    LD=     P1_input K3
      MOVP    K3 P1_output
      OUT     punch3
      MOVP    P3_input P3_output
      AND=    end_step_01 K3
      +P      K1 step_on
      MOVP    K0 end_step_01
      OUT     next_signal_03
86    LD=     P1_input K4
      MOVP    K4 P1_output
      OUT     punch4
      MOVP    P3_input P3_output
      AND=    end_step_01 K4
      +P      K1 step_on
      MOVP    K0 end_step_01
      OUT     next_signal_04
109   LD=     P1_input K5
      MOVP    K5 P1_output
      OUT     punch5
      MOVP    P3_input P3_output
      AND=    end_step_01 K5
      +P      K1 step_on
      MOVP    K0 end_step_01
      OUT     next_signal_05
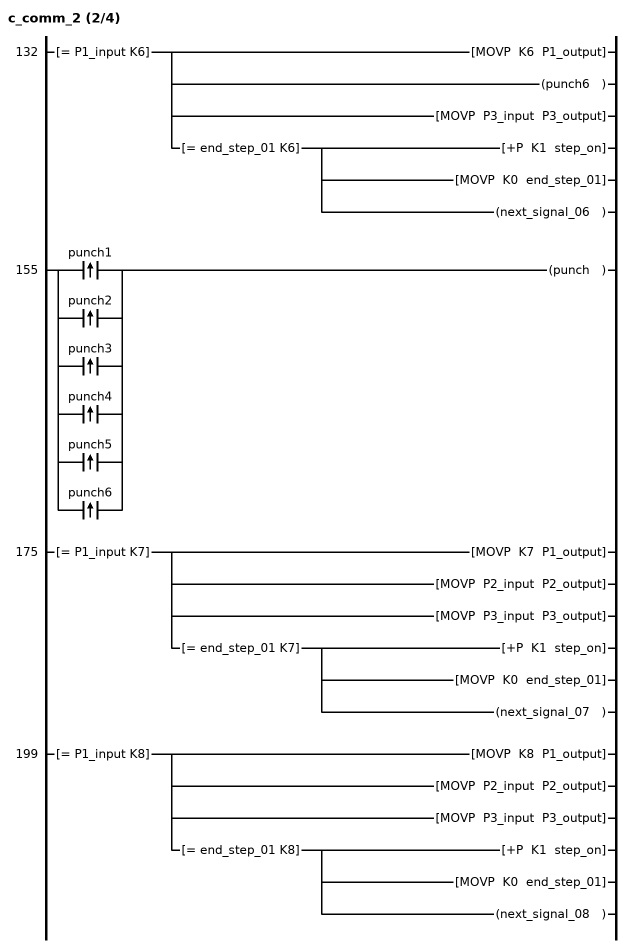
132   LD=     P1_input K6
      MOVP    K6 P1_output
      OUT     punch6
      MOVP    P3_input P3_output
      AND=    end_step_01 K6
      +P      K1 step_on
      MOVP    K0 end_step_01
      OUT     next_signal_06
155   LDP     punch1
      ORP     punch2
      ORP     punch3
      ORP     punch4
      ORP     punch5
      ORP     punch6
      OUT     punch
175   LD=     P1_input K7
      MOVP    K7 P1_output
      MOVP    P2_input P2_output
      MOVP    P3_input P3_output
      AND=    end_step_01 K7
      +P      K1 step_on
      MOVP    K0 end_step_01
      OUT     next_signal_07
199   LD=     P1_input K8
      MOVP    K8 P1_output
      MOVP    P2_input P2_output
      MOVP    P3_input P3_output
      AND=    end_step_01 K8
      +P      K1 step_on
      MOVP    K0 end_step_01
      OUT     next_signal_08
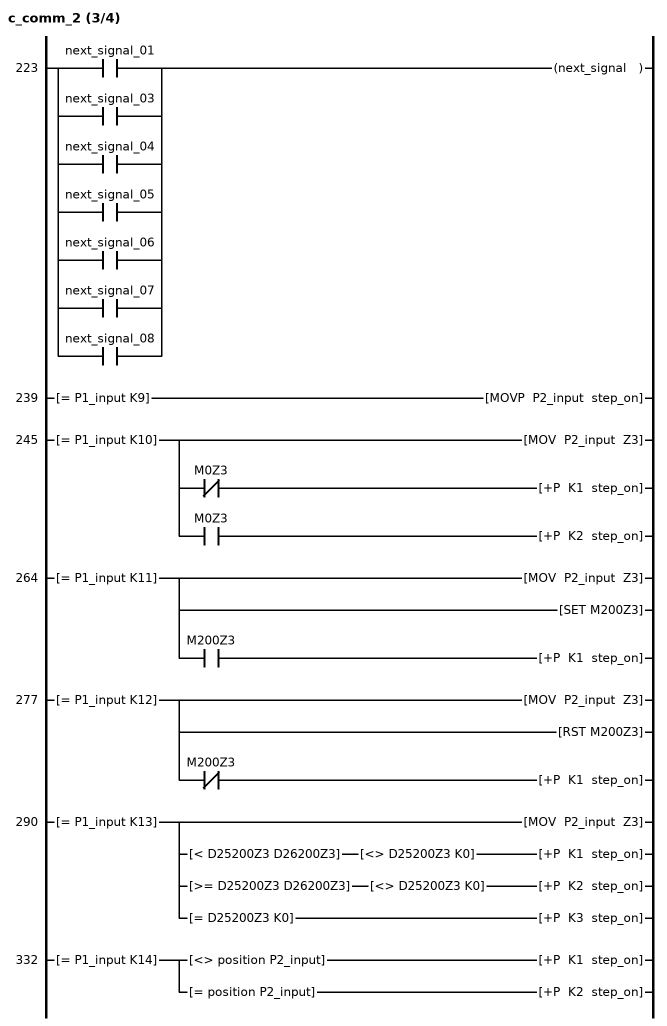
223   LD      next_signal_01
      OR      next_signal_03
      OR      next_signal_04
      OR      next_signal_05
      OR      next_signal_06
      OR      next_signal_07
      OR      next_signal_08
      OUT     next_signal
239   LD=     P1_input K9
      MOVP    P2_input step_on
245   LD=     P1_input K10
      MOV     P2_input Z3
      MPS
      ANI     M0Z3
      +P      K1 step_on
      MPP
      AND     M0Z3
      +P      K2 step_on
264   LD=     P1_input K11
      MOV     P2_input Z3
      SET     M200Z3
      AND     M200Z3
      +P      K1 step_on
277   LD=     P1_input K12
      MOV     P2_input Z3
      RST     M200Z3
      ANI     M200Z3
      +P      K1 step_on
290   LD=     P1_input K13
      MOV     P2_input Z3
      MPS
      AND<    D25200Z3 D26200Z3
      AND<>   D25200Z3 K0
      +P      K1 step_on
      MRD
      AND>=   D25200Z3 D26200Z3
      AND<>   D25200Z3 K0
      +P      K2 step_on
      MPP
      AND=    D25200Z3 K0
      +P      K3 step_on
332   LD=     P1_input K14
      MPS
      AND<>   position P2_input
      +P      K1 step_on
      MPP
      AND=    position P2_input
      +P      K2 step_on
